TYPE ST_SorterConfig :
STRUCT
	Name				: STRING[5];
	Length				: UINT;
	InductWindow		: UINT;
	MinimumLength		: UINT;
	TailEndLength 		: UINT;
	Output2Offset		: UINT;
	DefaultDestination 	: UINT;
	RecircDestination 	: UINT;
	RecircUsed			: BOOL;
	RetainOnRestart		: BOOL;
	DivertCount			: DINT;
END_STRUCT
END_TYPE

(* stored: Version 1.1.0.1, ProductVersion 3.1.4024.4
   DUT ST_SorterConfig: Id {9ce3f4df-7db1-4bfa-b8ac-5118da50235f} *)
